(* IEC 61131-3 sources: RL_MAR/experiments/comparison/llm4plc/results/gpt-4o_20260507_114630/20260507_120529, 4 files *)

(* ---- generated_code_iteration_0.st ---- *)
plaintext
START_ST
FUNCTION_BLOCK CarParkingSystem
VAR_INPUT
    NewCarSlot : INT; (* Input for new car arrival slot number *)
END_VAR
VAR_OUTPUT
    Elevator1Busy : BOOL; (* Elevator 1 status - busy or idle *)
    Elevator2Busy : BOOL; (* Elevator 2 status - busy or idle *)
    Elevator1Position : INT; (* Elevator 1 current position *)
    Elevator2Position : INT; (* Elevator 2 current position *)
END_VAR
VAR
    state : INT; (* Current state of the system *)
    Elevator1Target : INT; (* Target position for Elevator 1 *)
    Elevator2Target : INT; (* Target position for Elevator 2 *)
    CarSlots : ARRAY[1..100] OF BOOL; (* Array to represent parking slots - TRUE if occupied *)
    CurrentSlot : INT; (* Loop counter for scanning slots *)
END_VAR

(* Initialization of variables *)
IF NOT INIT THEN
    state := 0; (* Start in IDLE state *)
    Elevator1Busy := FALSE;
    Elevator2Busy := FALSE;
    Elevator1Position := 0;
    Elevator2Position := 0;
    Elevator1Target := 0;
    Elevator2Target := 0;
    FOR CurrentSlot := 1 TO 100 DO
        CarSlots[CurrentSlot] := FALSE; (* Initialize all slots as unoccupied *)
    END_FOR;
    INIT := TRUE;
END_IF;

(* State Machine *)
CASE state OF
    (* STATE 0: IDLE *)
    0:
        Elevator1Busy := FALSE;
        Elevator2Busy := FALSE;
        IF NewCarSlot > 0 THEN
            state := 1; (* Transition to ASSIGN ELEVATOR state *)
        END_IF;

    (* STATE 1: ASSIGN ELEVATOR *)
    1:
        IF (NewCarSlot >= 1 AND NewCarSlot <= 50) AND (Elevator1Busy = FALSE) THEN
            Elevator1Target := NewCarSlot;
            Elevator1Busy := TRUE;
            state := 2; (* Transition to MOVE ELEVATOR 1 state *)
        ELSIF (NewCarSlot >= 51 AND NewCarSlot <= 100) AND (Elevator2Busy = FALSE) THEN
            Elevator2Target := NewCarSlot;
            Elevator2Busy := TRUE;
            state := 3; (* Transition to MOVE ELEVATOR 2 state *)
        END_IF;

    (* STATE 2: MOVE ELEVATOR 1 *)
    2:
        IF Elevator1Position < Elevator1Target THEN
            Elevator1Position := Elevator1Position + 1; (* Move Elevator 1 up *)
        ELSIF Elevator1Position > Elevator1Target THEN
            Elevator1Position := Elevator1Position - 1; (* Move Elevator 1 down *)
        ELSE
            state := 4; (* Transition to UPDATE SLOT STATUS state *)
        END_IF;

    (* STATE 3: MOVE ELEVATOR 2 *)
    3:
        IF Elevator2Position < Elevator2Target THEN
            Elevator2Position := Elevator2Position + 1; (* Move Elevator 2 up *)
        ELSIF Elevator2Position > Elevator2Target THEN
            Elevator2Position := Elevator2Position - 1; (* Move Elevator 2 down *)
        ELSE
            state := 4; (* Transition to UPDATE SLOT STATUS state *)
        END_IF;

    (* STATE 4: UPDATE SLOT STATUS *)
    4:
        CarSlots[NewCarSlot] := TRUE; (* Mark the slot as occupied *)
        NewCarSlot := 0; (* Reset NewCarSlot to indicate task completion *)
        IF Elevator1Position = Elevator1Target THEN
            Elevator1Busy := FALSE; (* Mark Elevator 1 as idle *)
        END_IF;
        IF Elevator2Position = Elevator2Target THEN
            Elevator2Busy := FALSE; (* Mark Elevator 2 as idle *)
        END_IF;
        IF (Elevator1Busy = FALSE) AND (Elevator2Busy = FALSE) THEN
            state := 0; (* Transition back to IDLE state *)
        END_IF;
END_CASE;

END_FUNCTION_BLOCK
END_ST

(* ---- generated_code_iteration_1.st ---- *)
START_REASON
The feedback indicates that the Structured Text (ST) code failed the CODESYS compiler validation due to a type mismatch error. Specifically, the error message "此处需要有类型 'BOOL'的表达式" translates to "A 'BOOL' type expression is required here." This suggests that somewhere in the code, a condition or expression that requires a `BOOL` type is either missing or incorrectly specified.

Upon reviewing the code, the issue likely arises from the initialization of the `INIT` variable. The variable `INIT` is used in the initialization block but is not declared in the `VAR` section. Additionally, it is being used as a `BOOL` type without explicit declaration. This would cause the compiler to fail since `INIT` is not recognized as a `BOOL` type.

To resolve this, I will declare `INIT` as a `BOOL` variable in the `VAR` section and ensure it is properly initialized. This should address the type mismatch error and allow the code to pass validation.
END_REASON

START_ST
FUNCTION_BLOCK CarParkingSystem
VAR_INPUT
    NewCarSlot : INT; (* Input for new car arrival slot number *)
END_VAR
VAR_OUTPUT
    Elevator1Busy : BOOL; (* Elevator 1 status - busy or idle *)
    Elevator2Busy : BOOL; (* Elevator 2 status - busy or idle *)
    Elevator1Position : INT; (* Elevator 1 current position *)
    Elevator2Position : INT; (* Elevator 2 current position *)
END_VAR
VAR
    state : INT; (* Current state of the system *)
    Elevator1Target : INT; (* Target position for Elevator 1 *)
    Elevator2Target : INT; (* Target position for Elevator 2 *)
    CarSlots : ARRAY[1..100] OF BOOL; (* Array to represent parking slots - TRUE if occupied *)
    CurrentSlot : INT; (* Loop counter for scanning slots *)
    INIT : BOOL; (* Initialization flag *)
END_VAR

(* Initialization of variables *)
IF NOT INIT THEN
    state := 0; (* Start in IDLE state *)
    Elevator1Busy := FALSE;
    Elevator2Busy := FALSE;
    Elevator1Position := 0;
    Elevator2Position := 0;
    Elevator1Target := 0;
    Elevator2Target := 0;
    FOR CurrentSlot := 1 TO 100 DO
        CarSlots[CurrentSlot] := FALSE; (* Initialize all slots as unoccupied *)
    END_FOR;
    INIT := TRUE; (* Set initialization flag to TRUE *)
END_IF;

(* State Machine *)
CASE state OF
    (* STATE 0: IDLE *)
    0:
        Elevator1Busy := FALSE;
        Elevator2Busy := FALSE;
        IF NewCarSlot > 0 THEN
            state := 1; (* Transition to ASSIGN ELEVATOR state *)
        END_IF;

    (* STATE 1: ASSIGN ELEVATOR *)
    1:
        IF (NewCarSlot >= 1 AND NewCarSlot <= 50) AND (Elevator1Busy = FALSE) THEN
            Elevator1Target := NewCarSlot;
            Elevator1Busy := TRUE;
            state := 2; (* Transition to MOVE ELEVATOR 1 state *)
        ELSIF (NewCarSlot >= 51 AND NewCarSlot <= 100) AND (Elevator2Busy = FALSE) THEN
            Elevator2Target := NewCarSlot;
            Elevator2Busy := TRUE;
            state := 3; (* Transition to MOVE ELEVATOR 2 state *)
        END_IF;

    (* STATE 2: MOVE ELEVATOR 1 *)
    2:
        IF Elevator1Position < Elevator1Target THEN
            Elevator1Position := Elevator1Position + 1; (* Move Elevator 1 up *)
        ELSIF Elevator1Position > Elevator1Target THEN
            Elevator1Position := Elevator1Position - 1; (* Move Elevator 1 down *)
        ELSE
            state := 4; (* Transition to UPDATE SLOT STATUS state *)
        END_IF;

    (* STATE 3: MOVE ELEVATOR 2 *)
    3:
        IF Elevator2Position < Elevator2Target THEN
            Elevator2Position := Elevator2Position + 1; (* Move Elevator 2 up *)
        ELSIF Elevator2Position > Elevator2Target THEN
            Elevator2Position := Elevator2Position - 1; (* Move Elevator 2 down *)
        ELSE
            state := 4; (* Transition to UPDATE SLOT STATUS state *)
        END_IF;

    (* STATE 4: UPDATE SLOT STATUS *)
    4:
        CarSlots[NewCarSlot] := TRUE; (* Mark the slot as occupied *)
        NewCarSlot := 0; (* Reset NewCarSlot to indicate task completion *)
        IF Elevator1Position = Elevator1Target THEN
            Elevator1Busy := FALSE; (* Mark Elevator 1 as idle *)
        END_IF;
        IF Elevator2Position = Elevator2Target THEN
            Elevator2Busy := FALSE; (* Mark Elevator 2 as idle *)
        END_IF;
        IF (Elevator1Busy = FALSE) AND (Elevator2Busy = FALSE) THEN
            state := 0; (* Transition back to IDLE state *)
        END_IF;
END_CASE;

END_FUNCTION_BLOCK
END_ST

(* ---- generated_code_iteration_2.st ---- *)
START_REASON
The feedback indicates that the validation failed due to an encoding issue, specifically related to the 'gbk' codec. This error suggests that there are non-ASCII characters or unsupported characters in the code, which the compiler cannot process. Upon reviewing the code, the comments and variable descriptions contain non-ASCII characters (e.g., "此处需要有类型 'BOOL'的表达式" and possibly others). These characters are likely causing the encoding issue.

To fix this, I will ensure that all comments and text in the code are written in plain ASCII characters. Non-ASCII characters will be replaced with equivalent English text to maintain compatibility with the compiler. Additionally, I will review the code for any other potential issues and ensure it adheres to proper syntax and structure.
END_REASON

START_ST
FUNCTION_BLOCK CarParkingSystem
VAR_INPUT
    NewCarSlot : INT; (* Input for new car arrival slot number *)
END_VAR
VAR_OUTPUT
    Elevator1Busy : BOOL; (* Elevator 1 status - busy or idle *)
    Elevator2Busy : BOOL; (* Elevator 2 status - busy or idle *)
    Elevator1Position : INT; (* Elevator 1 current position *)
    Elevator2Position : INT; (* Elevator 2 current position *)
END_VAR
VAR
    state : INT; (* Current state of the system *)
    Elevator1Target : INT; (* Target position for Elevator 1 *)
    Elevator2Target : INT; (* Target position for Elevator 2 *)
    CarSlots : ARRAY[1..100] OF BOOL; (* Array to represent parking slots - TRUE if occupied *)
    CurrentSlot : INT; (* Loop counter for scanning slots *)
    INIT : BOOL; (* Initialization flag *)
END_VAR

(* Initialization of variables *)
IF NOT INIT THEN
    state := 0; (* Start in IDLE state *)
    Elevator1Busy := FALSE;
    Elevator2Busy := FALSE;
    Elevator1Position := 0;
    Elevator2Position := 0;
    Elevator1Target := 0;
    Elevator2Target := 0;
    FOR CurrentSlot := 1 TO 100 DO
        CarSlots[CurrentSlot] := FALSE; (* Initialize all slots as unoccupied *)
    END_FOR;
    INIT := TRUE; (* Set initialization flag to TRUE *)
END_IF;

(* State Machine *)
CASE state OF
    (* STATE 0: IDLE *)
    0:
        Elevator1Busy := FALSE;
        Elevator2Busy := FALSE;
        IF NewCarSlot > 0 THEN
            state := 1; (* Transition to ASSIGN ELEVATOR state *)
        END_IF;

    (* STATE 1: ASSIGN ELEVATOR *)
    1:
        IF (NewCarSlot >= 1 AND NewCarSlot <= 50) AND (Elevator1Busy = FALSE) THEN
            Elevator1Target := NewCarSlot;
            Elevator1Busy := TRUE;
            state := 2; (* Transition to MOVE ELEVATOR 1 state *)
        ELSIF (NewCarSlot >= 51 AND NewCarSlot <= 100) AND (Elevator2Busy = FALSE) THEN
            Elevator2Target := NewCarSlot;
            Elevator2Busy := TRUE;
            state := 3; (* Transition to MOVE ELEVATOR 2 state *)
        END_IF;

    (* STATE 2: MOVE ELEVATOR 1 *)
    2:
        IF Elevator1Position < Elevator1Target THEN
            Elevator1Position := Elevator1Position + 1; (* Move Elevator 1 up *)
        ELSIF Elevator1Position > Elevator1Target THEN
            Elevator1Position := Elevator1Position - 1; (* Move Elevator 1 down *)
        ELSE
            state := 4; (* Transition to UPDATE SLOT STATUS state *)
        END_IF;

    (* STATE 3: MOVE ELEVATOR 2 *)
    3:
        IF Elevator2Position < Elevator2Target THEN
            Elevator2Position := Elevator2Position + 1; (* Move Elevator 2 up *)
        ELSIF Elevator2Position > Elevator2Target THEN
            Elevator2Position := Elevator2Position - 1; (* Move Elevator 2 down *)
        ELSE
            state := 4; (* Transition to UPDATE SLOT STATUS state *)
        END_IF;

    (* STATE 4: UPDATE SLOT STATUS *)
    4:
        CarSlots[NewCarSlot] := TRUE; (* Mark the slot as occupied *)
        NewCarSlot := 0; (* Reset NewCarSlot to indicate task completion *)
        IF Elevator1Position = Elevator1Target THEN
            Elevator1Busy := FALSE; (* Mark Elevator 1 as idle *)
        END_IF;
        IF Elevator2Position = Elevator2Target THEN
            Elevator2Busy := FALSE; (* Mark Elevator 2 as idle *)
        END_IF;
        IF (Elevator1Busy = FALSE) AND (Elevator2Busy = FALSE) THEN
            state := 0; (* Transition back to IDLE state *)
        END_IF;
END_CASE;

END_FUNCTION_BLOCK
END_ST

(* ---- generated_code_iteration_3.st ---- *)
START_REASON
The feedback indicates that the validation failed due to an encoding issue, specifically related to the 'gbk' codec. This issue is caused by non-ASCII characters in the code, which the compiler cannot process. Upon reviewing the provided code, it appears that all comments and variable descriptions are already in English and do not contain non-ASCII characters. However, the issue might stem from hidden or invisible non-ASCII characters (e.g., spaces, line breaks, or other formatting artifacts) introduced during editing or copying.

To resolve this issue, I will:
1. Remove any potential hidden non-ASCII characters by retyping the code in a plain text editor that ensures ASCII encoding.
2. Ensure all comments, variable names, and descriptions are in plain ASCII characters.
3. Revalidate the code structure and syntax to ensure compliance with the Structured Text (ST) language.

I will now rewrite the code to ensure it is free of encoding issues and adheres to the correct syntax.
END_REASON

START_ST
FUNCTION_BLOCK CarParkingSystem
VAR_INPUT
    NewCarSlot : INT; (* Input for new car arrival slot number *)
END_VAR
VAR_OUTPUT
    Elevator1Busy : BOOL; (* Elevator 1 status - busy or idle *)
    Elevator2Busy : BOOL; (* Elevator 2 status - busy or idle *)
    Elevator1Position : INT; (* Elevator 1 current position *)
    Elevator2Position : INT; (* Elevator 2 current position *)
END_VAR
VAR
    state : INT; (* Current state of the system *)
    Elevator1Target : INT; (* Target position for Elevator 1 *)
    Elevator2Target : INT; (* Target position for Elevator 2 *)
    CarSlots : ARRAY[1..100] OF BOOL; (* Array to represent parking slots - TRUE if occupied *)
    CurrentSlot : INT; (* Loop counter for scanning slots *)
    INIT : BOOL; (* Initialization flag *)
END_VAR

(* Initialization of variables *)
IF NOT INIT THEN
    state := 0; (* Start in IDLE state *)
    Elevator1Busy := FALSE;
    Elevator2Busy := FALSE;
    Elevator1Position := 0;
    Elevator2Position := 0;
    Elevator1Target := 0;
    Elevator2Target := 0;
    FOR CurrentSlot := 1 TO 100 DO
        CarSlots[CurrentSlot] := FALSE; (* Initialize all slots as unoccupied *)
    END_FOR;
    INIT := TRUE; (* Set initialization flag to TRUE *)
END_IF;

(* State Machine *)
CASE state OF
    (* STATE 0: IDLE *)
    0:
        Elevator1Busy := FALSE;
        Elevator2Busy := FALSE;
        IF NewCarSlot > 0 THEN
            state := 1; (* Transition to ASSIGN ELEVATOR state *)
        END_IF;

    (* STATE 1: ASSIGN ELEVATOR *)
    1:
        IF (NewCarSlot >= 1 AND NewCarSlot <= 50) AND (Elevator1Busy = FALSE) THEN
            Elevator1Target := NewCarSlot;
            Elevator1Busy := TRUE;
            state := 2; (* Transition to MOVE ELEVATOR 1 state *)
        ELSIF (NewCarSlot >= 51 AND NewCarSlot <= 100) AND (Elevator2Busy = FALSE) THEN
            Elevator2Target := NewCarSlot;
            Elevator2Busy := TRUE;
            state := 3; (* Transition to MOVE ELEVATOR 2 state *)
        END_IF;

    (* STATE 2: MOVE ELEVATOR 1 *)
    2:
        IF Elevator1Position < Elevator1Target THEN
            Elevator1Position := Elevator1Position + 1; (* Move Elevator 1 up *)
        ELSIF Elevator1Position > Elevator1Target THEN
            Elevator1Position := Elevator1Position - 1; (* Move Elevator 1 down *)
        ELSE
            state := 4; (* Transition to UPDATE SLOT STATUS state *)
        END_IF;

    (* STATE 3: MOVE ELEVATOR 2 *)
    3:
        IF Elevator2Position < Elevator2Target THEN
            Elevator2Position := Elevator2Position + 1; (* Move Elevator 2 up *)
        ELSIF Elevator2Position > Elevator2Target THEN
            Elevator2Position := Elevator2Position - 1; (* Move Elevator 2 down *)
        ELSE
            state := 4; (* Transition to UPDATE SLOT STATUS state *)
        END_IF;

    (* STATE 4: UPDATE SLOT STATUS *)
    4:
        CarSlots[NewCarSlot] := TRUE; (* Mark the slot as occupied *)
        NewCarSlot := 0; (* Reset NewCarSlot to indicate task completion *)
        IF Elevator1Position = Elevator1Target THEN
            Elevator1Busy := FALSE; (* Mark Elevator 1 as idle *)
        END_IF;
        IF Elevator2Position = Elevator2Target THEN
            Elevator2Busy := FALSE; (* Mark Elevator 2 as idle *)
        END_IF;
        IF (Elevator1Busy = FALSE) AND (Elevator2Busy = FALSE) THEN
            state := 0; (* Transition back to IDLE state *)
        END_IF;
END_CASE;

END_FUNCTION_BLOCK
END_ST
